(* IEC 61131-3 sources: com.logicals.lc3.webinar/usRTS_RPMControl_iSOC/src_FB_LIB_SAFE/Safe/PLCOpen (part 3) *)

(* ---- SF_PSE.iecst ---- *)
USING logicals.web.standard.safe;

NAMESPACE logicals.web.standard.safe
NAMESPACE plcopen

/*
 * This function block is a safety-related function block for monitoring Pressure-Sensitive-Equipment (PSE) like Safety Mats, Bumper etc.
 */
FUNCTION_BLOCK SF_PSE
	{ altName:="SF_PSE"; bgColor:="Gold"; width:=320; }
	VAR_INPUT
		/* See Section 5.1.1 General Input Parameters */
		Activate : BOOL := FALSE;
		/* Safety demand input.
		 * Variable.
		 * FALSE: PSE actuated, demand for safety-related response.
		 * TRUE: PSE not actuated, no demand for safety-related response.
		 * Safety control system must be able to detect a very short interruption of the PSE
		 * (which is specified in EN 1760: minimum 200 ms), when the PSE is used in applications as a safety device.
		 */
		S_PSE_In : SAFEBOOL := SAFEBOOL_Constant#SAFEFALSE;
		/* See Section 5.1.1 General Input Parameters */
		S_StartReset : SAFEBOOL := SAFEBOOL_Constant#SAFEFALSE;
		/* See Section 5.1.1 General Input Parameters */
		S_AutoReset : SAFEBOOL := SAFEBOOL_Constant#SAFEFALSE;
		/* See Section 5.1.1 General Input Parameters */
		Reset : BOOL := FALSE;
	END_VAR
	VAR_OUTPUT
		/* See Section 5.1.2 General Output Parameters */
		Ready : BOOL := FALSE;
		/* Output for the safety-related response.
		 * FALSE: Safety output disabled. Demand for safety-related response (e.g., reset requested or internal errors active).
		 * TRUE: Safety output enabled. No demand for safety-related response.
		 */
		S_PSE_Out : SAFEBOOL := SAFEBOOL_Constant#SAFEFALSE;
		/* Optional. See 5.1.2 General Output Parameters */
		SafetyDemand : BOOL := FALSE;
		/* Optional. See 5.1.2 General Output Parameters */
		ResetRequest : BOOL := FALSE;
		/* See Section 5.1.2 General Output Parameters */
		Error : BOOL := FALSE;
		/* See Section 5.1.2 General Output Parameters */
		DiagCode : WORD := 16#0000;
	END_VAR
	VAR
		GenericSafetyDemand : SFB_GenericSafetyDemand;
	END_VAR

	GenericSafetyDemand(
		Activate := Activate,
		S_SafetyDemandIn := S_PSE_In,
		S_StartReset := S_StartReset,
		S_AutoReset := S_AutoReset,
		Reset := Reset,
		Ready => Ready,
		S_SafetyDemandOut => S_PSE_Out,
		SafetyDemand => SafetyDemand,
		ResetRequest => ResetRequest,
		Error => Error,
		DiagCode => DiagCode,
		ENO => ENO
	);

END_FUNCTION_BLOCK

END_NAMESPACE
END_NAMESPACE

(* ---- SF_ResetButton.iecst ---- *)
USING logicals.web.standard.safe;

NAMESPACE logicals.web.standard.safe
NAMESPACE plcopen

TYPE
	SF_ResetButton_State : UINT(
	/* TrailingMinimum > TrailingMaximum OR TrailingMinimum < 100 msec. */
	Parameter_Error := 16#C000,
	/* ResetIn is TRUE while waiting for NOT ResetIn. */
	Reset_Error := 16#C001,
	/* TrailingMaximum elapsed before detecting F_TRIG at ResetIn. Waiting for R_TRIG at ResetIn. */
	Error_Trailing_Maximum := 16#C3E0,
	/* F_TRIG at ResetIn detected before TrailingMinimum elapsed. Waiting for R_TRIG at ResetIn. */
	Error_Trailing_Minimum := 16#C3F0,
	/* The function block is not active (initial state). */
	Idle := 16#0000,
	/* The function block is enabled. Wait for R_TRIG at ResetIn. */
	Wait_for_R_TRIG := 16#83E2,
	/* ResetIn is TRUE. Wait for F_TRIG at ResetIn */
	Wait_for_F_TRIG := 16#83F2,
	/* Valid reset behavior was detected. The state is valid for at least one cycle and will automatically transfer to 83E2. */
	Reset_Detected := 16#8000
	);
END_TYPE

/*
 * This function block adds the trailing edge functionality to all the function blocks with reset input with rising edge detection. This can be used to comply to EN ISO 13849-1:2015
 */
FUNCTION_BLOCK SF_ResetButton
	{ altName:="SF_ResetButton"; bgColor:="Gold"; width:=380; }
	VAR_INPUT
		/* Input which should be connected to the ResetRequest output of the paired FB.
			TRUE: ResetRequested
			FALSE: No reset requested / no monitoring of ResetIn. */
		ResetRequested : BOOL := TRUE;
		/* Variable.
			Input of reset button
			FALSE: reset button released;
			TRUE: reset button actuated by operator. */
		Button : BOOL := FALSE;
		/* Constant. Valid in trailing mode. Minimum time that the reset switch has to be actuated.
			If the reset button is pushed shorter than this time, the reset is ignored.
			Typical value 350msec.Absolut minimum value is 100msec.Minimum value 2 PLC cycles. */
		TrailingMinimum : TIME := T#350ms;
		/* Constant. Valid in trailing mode.
			Maximum time that the reset switch is actuated.
			Typical value can be around 2 sec. If the reset button is pushed longer than this time, the reset is ignored. */
		TrailingMaximum : TIME := T#2s;
	END_VAR
	VAR_OUTPUT
		/* See 5.1.2 General Output Parameters */
		Ready : BOOL := FALSE;
		/* Pulse for the initiation of the reset procedure.
			This pulse is generated after the falling edge.
			Pulse output with rising edge first. At least 1 cycle. */
		ResetOut : BOOL := FALSE;
		/* See 5.1.2 General Output Parameters */
		Error : BOOL := FALSE;
		/* See 5.1.2 General Output Parameters */
		DiagCode : WORD := 16#0000;
	END_VAR
	VAR
		TrailingMinimumTimer : TON;
		TrailingMaximumTimer : TON;
		R_Trig_Button : R_TRIG;
		F_Trig_Button : F_TRIG;
	END_VAR

	R_Trig_Button(Button);
	F_Trig_Button(Button);

	IF(NOT ResetRequested) THEN
		DiagCode := TO_WORD(SF_ResetButton_State#Idle);
	ELSE
		CASE TO_UINT(DiagCode) OF
			SF_ResetButton_State#Idle:
				/* IF(ResetRequested) THEN - ResetRequested is always true here */
					IF(Button) THEN
						DiagCode := TO_WORD(SF_ResetButton_State#Reset_Error);
					ELSE
					DiagCode := TO_WORD(SF_ResetButton_State#Wait_for_R_TRIG);
					END_IF;
			SF_ResetButton_State#Wait_for_R_TRIG:
				IF(TrailingMinimum > TrailingMaximum) OR (TrailingMinimum < T#100ms) THEN
					DiagCode := TO_WORD(SF_ResetButton_State#Parameter_Error);
				ELSIF(R_Trig_Button.Q) THEN
					DiagCode := TO_WORD(SF_ResetButton_State#Wait_for_F_TRIG);
				END_IF;
			SF_ResetButton_State#Reset_Error:
				IF(NOT Button) THEN
					DiagCode := TO_WORD(SF_ResetButton_State#Wait_for_R_TRIG);
				END_IF;
			SF_ResetButton_State#Wait_for_F_TRIG:
				TrailingMinimumTimer();
				TrailingMaximumTimer();
				IF(F_Trig_Button.Q) AND (NOT TrailingMinimumTimer.Q) THEN
					DiagCode := TO_WORD(SF_ResetButton_State#Error_Trailing_Minimum);
				ELSIF(TrailingMaximumTimer.Q) THEN
					DiagCode := TO_WORD(SF_ResetButton_State#Error_Trailing_Maximum);
				ELSIF(F_Trig_Button.Q) THEN
					DiagCode := TO_WORD(SF_ResetButton_State#Reset_Detected);
				END_IF;
			SF_ResetButton_State#Error_Trailing_Maximum:
				IF(R_Trig_Button.Q) THEN
					DiagCode := TO_WORD(SF_ResetButton_State#Wait_for_F_TRIG);
				END_IF;
			SF_ResetButton_State#Error_Trailing_Minimum:
				IF(R_Trig_Button.Q) THEN
					DiagCode := TO_WORD(SF_ResetButton_State#Wait_for_F_TRIG);
				END_IF;
			SF_ResetButton_State#Reset_Detected:
				DiagCode := TO_WORD(SF_ResetButton_State#Wait_for_R_TRIG);
			ELSE
				ENO := FALSE;
		END_CASE;
	END_IF;

		CASE TO_UINT(DiagCode) OF
			SF_ResetButton_State#Parameter_Error:
				TrailingMinimumTimer(IN := FALSE);
				TrailingMaximumTimer(IN := FALSE);
				Ready := TRUE;
				ResetOut := FALSE;
				Error := TRUE;
			SF_ResetButton_State#Reset_Error:
				TrailingMinimumTimer(IN := FALSE);
				TrailingMaximumTimer(IN := FALSE);
				Ready := TRUE;
				ResetOut := FALSE;
				Error := TRUE;
			SF_ResetButton_State#Error_Trailing_Maximum:
				TrailingMinimumTimer(IN := FALSE);
				TrailingMaximumTimer(IN := FALSE);
				Ready := TRUE;
				ResetOut := FALSE;
				Error := TRUE;
			SF_ResetButton_State#Error_Trailing_Minimum:
				TrailingMinimumTimer(IN := FALSE);
				TrailingMaximumTimer(IN := FALSE);
				Ready := TRUE;
				ResetOut := FALSE;
				Error := TRUE;
			SF_ResetButton_State#Idle:
				TrailingMinimumTimer(IN := FALSE);
				TrailingMaximumTimer(IN := FALSE);
				Ready := FALSE;
				ResetOut := FALSE;
				Error := FALSE;
			SF_ResetButton_State#Wait_for_R_TRIG:
				TrailingMinimumTimer(IN := FALSE);
				TrailingMaximumTimer(IN := FALSE);
				Ready := TRUE;
				ResetOut := FALSE;
				Error := FALSE;
			SF_ResetButton_State#Wait_for_F_TRIG:
				TrailingMinimumTimer(IN := TRUE, PT := TrailingMinimum);
				TrailingMaximumTimer(IN := TRUE, PT := TrailingMaximum);
				Ready := TRUE;
				ResetOut := FALSE;
				Error := FALSE;
			SF_ResetButton_State#Reset_Detected:
				TrailingMinimumTimer(IN := FALSE);
				TrailingMaximumTimer(IN := FALSE);
				Ready := TRUE;
				ResetOut := TRUE;
				Error := FALSE;
			ELSE
				ENO := FALSE;
		END_CASE;
END_FUNCTION_BLOCK

END_NAMESPACE
END_NAMESPACE

(* ---- SF_SafetyRequest.iecst ---- *)
USING logicals.web.standard.safe;

NAMESPACE logicals.web.standard.safe
NAMESPACE plcopen

TYPE
	SF_SafetyRequest_State : UINT(
	/* Acknowledgment lost while in the Safe state. */
	Acknowledge_Lost := 16#C010,
	/* S_OpMode request could not be completed within the monitoring time. */
	MonitoringTime_Elapsed := 16#C020,
	/* Static Reset detected in state 8401 (Init). */
	Reset_Error_1 := 16#C001,
	/* Static Reset detected in state C010 (Acknowledge Lost). */
	Reset_Error_2 := 16#C014,
	/* Static Reset detected in state C020 (MonitoringTime Elapsed). */
	Reset_Error_3 := 16#C011,
	/* The function block is not active (initial state). */
	Idle := 16#0000,
	/* Actuator is in a safe mode. */
	Safe_Mode:= 16#8000,
	/* State after Activate is set to TRUE or after a rising trigger at Reset. */
	Init := 16#8401,
	/* Operation mode without Acknowledge of safe mode */
	Operation_Mode:= 16#8802,
	/* Operation mode with Acknowledge of safe mode */
	Wait_For_Confirmation_OpMode := 16#8804,
	/* Waiting for confirmation from the drive (system interface). */
	Wait_For_Confirmation := 16#8002,
	/* Error was removed.
	* However S_OpMode must be set to TRUE or S_Acknowledge must become TRUE before the FB can be continued. */
	Wait_For_OpMode := 16#8004
	);
END_TYPE

/*
 * This function block provides the interface to a generic actuator, e.g. a safety drive or safety valve, to place the actuator in a safe state.
 */
FUNCTION_BLOCK SF_SafetyRequest
	{ altName:="SF_SafetyRequest"; bgColor:="Gold"; width:=400; }
	VAR_INPUT
		/* See Section 5.1.1 General Input Parameters */
		Activate : BOOL := FALSE;
		/* Variable.
		 * Requested mode of a generic safe actuator.
		 * FALSE: Safe mode is requested.
		 * TRUE: Operation mode is requested. */
		S_OpMode : SAFEBOOL := SAFEBOOL_Constant#SAFEFALSE;
		/* Variable.
		 * Confirmation of the generic actuator, if actuator is in the Safe state.
		 * FALSE: Operation mode (non-safe).
		 * TRUE: Safe mode. */
		S_Acknowledge : SAFEBOOL := SAFEBOOL_Constant#SAFEFALSE;
		/* Constant.
		 * Monitoring of the response time between the safety function request (S_OpMode set to FALSE)
		 * and the actuator acknowledgment (S_Acknowledge switches to TRUE). */
		MonitoringTime : TIME := T#0s;
		/* See Section 5.1.1 General Input Parameters */
		S_StartReset : SAFEBOOL := SAFEBOOL_Constant#SAFEFALSE;
		/* See Section 5.1.1 General Input Parameters with the functionality as an error removed acknowledge */
		Reset : BOOL := FALSE;
	END_VAR

	VAR_OUTPUT
		/* See Section 5.1.2 General Output Parameters */
		Ready : BOOL := FALSE;
		/* Confirmation of the Safe state.
		 * FALSE: Non-safe state.
		 * TRUE: Safe state. */
		S_SafetyActive : SAFEBOOL := SAFEBOOL_Constant#SAFEFALSE;
		/* Request to place the actuator in a safe state.
		 * FALSE: Safe state is requested.
		 * TRUE: Non-safe state. */
		S_SafetyRequest : SAFEBOOL := SAFEBOOL_Constant#SAFEFALSE;
		/* See Section 5.1.2 General Output Parameters */
		SafetyDemand : BOOL := FALSE;
		/* See Section 5.1.2 General Output Parameters */
		ResetRequest : BOOL := FALSE;
		/* See Section 5.1.2 General Output Parameters */
		Error : BOOL := FALSE;
		/* See Section 5.1.2 General Output Parameters */
		DiagCode : WORD := 16#0000;
	END_VAR

	VAR
		MonitoringTimer : TON;
		R_Trig_Reset : R_TRIG;
	END_VAR

	R_Trig_Reset(Reset);

	IF(NOT Activate) THEN
		DiagCode := TO_WORD(SF_SafetyRequest_State#Idle);
	ELSE
		CASE TO_UINT(DiagCode) OF
			SF_SafetyRequest_State#Idle:
				/* IF(Activate) THEN - ResetRequested is always true here */
					DiagCode := TO_WORD(SF_SafetyRequest_State#Init);
			SF_SafetyRequest_State#Init:
				IF(Reset AND NOT R_Trig_Reset.Q) THEN
					DiagCode := TO_WORD(SF_SafetyRequest_State#Reset_Error_1);
				ELSIF(R_Trig_Reset.Q AND IS_NOT(S_Acknowledge)) THEN
					DiagCode := TO_WORD(SF_SafetyRequest_State#Operation_Mode);
				ELSIF(R_Trig_Reset.Q AND IS(S_Acknowledge)) THEN
					DiagCode := TO_WORD(SF_SafetyRequest_State#Wait_For_Confirmation_OpMode);
				END_IF;
			SF_SafetyRequest_State#Operation_Mode:
				IF(IS_NOT(S_OpMode)) THEN
					DiagCode := TO_WORD(SF_SafetyRequest_State#Wait_For_Confirmation);
				ELSIF(IS(S_Acknowledge)) THEN
					DiagCode := TO_WORD(SF_SafetyRequest_State#Wait_For_Confirmation_OpMode);
				END_IF;
			SF_SafetyRequest_State#Wait_For_Confirmation_OpMode:
				IF(IS_NOT(S_Acknowledge)) THEN
					DiagCode := TO_WORD(SF_SafetyRequest_State#Operation_Mode);
				ELSIF(IS_NOT(S_OpMode)) THEN
					DiagCode := TO_WORD(SF_SafetyRequest_State#Wait_For_Confirmation);
				END_IF;
			SF_SafetyRequest_State#Wait_For_Confirmation:
				MonitoringTimer();
				IF(MonitoringTimer.Q) THEN
					DiagCode := TO_WORD(SF_SafetyRequest_State#MonitoringTime_Elapsed);
				ELSIF(IS(S_OpMode)) THEN
					DiagCode := TO_WORD(SF_SafetyRequest_State#Wait_For_Confirmation_OpMode);
				ELSIF(IS(S_Acknowledge)) THEN
					DiagCode := TO_WORD(SF_SafetyRequest_State#Safe_Mode);
				END_IF;
			SF_SafetyRequest_State#MonitoringTime_Elapsed:
				IF(Reset AND NOT R_Trig_Reset.Q) THEN
					DiagCode := TO_WORD(SF_SafetyRequest_State#Reset_Error_3);
				ELSIF(R_Trig_Reset.Q) THEN
					DiagCode := TO_WORD(SF_SafetyRequest_State#Wait_For_OpMode);
				END_IF;
			SF_SafetyRequest_State#Wait_For_OpMode:
				IF(IS(S_OpMode)) THEN
					DiagCode := TO_WORD(SF_SafetyRequest_State#Wait_For_Confirmation_OpMode);
				END_IF;
			SF_SafetyRequest_State#Safe_Mode:
				IF(IS_NOT(S_Acknowledge)) THEN
					DiagCode := TO_WORD(SF_SafetyRequest_State#Acknowledge_Lost);
				ELSIF(IS(S_OpMode)) THEN
					DiagCode := TO_WORD(SF_SafetyRequest_State#Wait_For_Confirmation_OpMode);
				END_IF;
			SF_SafetyRequest_State#Acknowledge_Lost:
				IF(Reset AND NOT R_Trig_Reset.Q) THEN
					DiagCode := TO_WORD(SF_SafetyRequest_State#Reset_Error_2);
				ELSIF(R_Trig_Reset.Q) THEN
					DiagCode := TO_WORD(SF_SafetyRequest_State#Wait_For_OpMode);
				END_IF;
			SF_SafetyRequest_State#Reset_Error_1:
				IF(NOT Reset) THEN
					DiagCode := TO_WORD(SF_SafetyRequest_State#Init);
				END_IF;
			SF_SafetyRequest_State#Reset_Error_2:
				IF(NOT Reset) THEN
					DiagCode := TO_WORD(SF_SafetyRequest_State#Acknowledge_Lost);
				END_IF;
			SF_SafetyRequest_State#Reset_Error_3:
				IF(NOT Reset) THEN
					DiagCode := TO_WORD(SF_SafetyRequest_State#MonitoringTime_Elapsed);
				END_IF;
		END_CASE;
	END_IF;

	CASE TO_UINT(DiagCode) OF
		SF_SafetyRequest_State#Idle:
			MonitoringTimer(IN := FALSE);
			Ready := FALSE;
			S_SafetyActive := SAFEBOOL_Constant#SAFEFALSE;
			S_SafetyRequest := SAFEBOOL_Constant#SAFEFALSE;
			SafetyDemand := FALSE;
			ResetRequest := FALSE;
			Error := FALSE;
		SF_SafetyRequest_State#Safe_Mode:
			MonitoringTimer(IN := FALSE);
			Ready := TRUE;
			S_SafetyActive := SAFEBOOL_Constant#SAFETRUE;
			S_SafetyRequest := SAFEBOOL_Constant#SAFEFALSE;
			SafetyDemand := FALSE;
			ResetRequest := FALSE;
			Error := FALSE;
		SF_SafetyRequest_State#Init:
			MonitoringTimer(IN := FALSE);
			Ready := TRUE;
			S_SafetyActive := SAFEBOOL_Constant#SAFEFALSE;
			S_SafetyRequest := SAFEBOOL_Constant#SAFEFALSE;
			SafetyDemand := FALSE;
			ResetRequest := TRUE;
			Error := FALSE;
		SF_SafetyRequest_State#Operation_Mode:
			MonitoringTimer(IN := FALSE);
			Ready := TRUE;
			S_SafetyActive := SAFEBOOL_Constant#SAFEFALSE;
			S_SafetyRequest := SAFEBOOL_Constant#SAFETRUE;
			SafetyDemand := TRUE;
			ResetRequest := FALSE;
			Error := FALSE;
		SF_SafetyRequest_State#Wait_For_Confirmation_OpMode:
			MonitoringTimer(IN := TRUE, PT := MonitoringTime);
			Ready := TRUE;
			S_SafetyActive := SAFEBOOL_Constant#SAFEFALSE;
			S_SafetyRequest := SAFEBOOL_Constant#SAFETRUE;
			SafetyDemand := TRUE;
			ResetRequest := FALSE;
			Error := FALSE;
		SF_SafetyRequest_State#Wait_For_Confirmation,
		SF_SafetyRequest_State#Wait_For_OpMode:
			MonitoringTimer(IN := TRUE, PT := MonitoringTime);
			Ready := TRUE;
			S_SafetyActive := SAFEBOOL_Constant#SAFEFALSE;
			S_SafetyRequest := SAFEBOOL_Constant#SAFEFALSE;
			SafetyDemand := FALSE;
			ResetRequest := FALSE;
			Error := FALSE;
		SF_SafetyRequest_State#Acknowledge_Lost,
		SF_SafetyRequest_State#MonitoringTime_Elapsed:
			MonitoringTimer(IN := FALSE);
			Ready := TRUE;
			S_SafetyActive := SAFEBOOL_Constant#SAFEFALSE;
			S_SafetyRequest := SAFEBOOL_Constant#SAFEFALSE;
			SafetyDemand := FALSE;
			ResetRequest := TRUE;
			Error := TRUE;
		SF_SafetyRequest_State#Reset_Error_1,
		SF_SafetyRequest_State#Reset_Error_2,
		SF_SafetyRequest_State#Reset_Error_3:
			MonitoringTimer(IN := FALSE);
			Ready := TRUE;
			S_SafetyActive := SAFEBOOL_Constant#SAFEFALSE;
			S_SafetyRequest := SAFEBOOL_Constant#SAFEFALSE;
			SafetyDemand := FALSE;
			ResetRequest := FALSE;
			Error := TRUE;
		ELSE
			ENO := FALSE;
	END_CASE;

	ENO := ENO AND CheckSAFEBOOL(S_OpMode) AND CheckSAFEBOOL(S_Acknowledge) AND CheckSAFEBOOL(S_StartReset);

END_FUNCTION_BLOCK

END_NAMESPACE
END_NAMESPACE

(* ---- SF_TestableSafetySensor.iecst ---- *)
USING logicals.web.standard.safe;

NAMESPACE logicals.web.standard.safe
NAMESPACE plcopen

TYPE
	SF_TestableSafetySensor_State : UINT(
	/* Invalid value at the TestTime parameter. Values between 0 ms and 150 ms are possible. */
	Parameter_Error := 16#C000,
	/* Static Reset condition detected after FB activation. */
	Reset_Error_1 := 16#C001,
	/* Static Reset condition detected in state 8403. */
	Reset_Error_2 := 16#C011,
	/* Static Reset condition detected in state Cx10. */
	Reset_Error_3 := 16#C021,
	/* Static Reset condition detected in state 8406. */
	Reset_Error_4 := 16#C031,
	/* Static Reset condition detected in state C000. */
	Reset_Error_5 := 16#C041,
	/* Static Reset condition detected in state 8413. */
	Reset_Error_6 := 16#C051,
	/* Test time elapsed in state 8020 or 8030. IF S_OSSD_IN = TRUE AND NoExternalTest = TRUE THEN x=4 ELSE x=0; */
	Test_Error_1 := 16#C410,
	Test_Error_2 := 16#C010,
	/* The function block is not active (initial state). */
	Idle := 16#0000,
	/* An activation has been detected by the FB. */
	Init := 16#8401,
	/* The FB has detected a safety demand. The switch has not been automatically tested yet. */
	ESPE_Interrupted_1 := 16#8802,
	/* Wait for rising trigger of Reset after state 8802. */
	Wait_for_Reset_1 := 16#8402,
	/* The automatic sensor test was faulty. An external manual sensor test is necessary.
	 * The support for the necessary external manual sensor test has been activated at the FB (NoExternalTest = FALSE).
	 * A negative signal edge at the sensor is required.
	 */
	External_Function_Test := 16#8002,
	/* The automatic sensor test was faulty. An external manual sensor test is necessary.
	 * The support for the necessary external manual sensor test has been activated at the FB (NoExternalTest = FALSE).
	 * A TRUE signal at the sensor is required.
	 */
	ESPE_Interrupted_External_Test := 16#8804,
	/* The automatic sensor test was faulty. An external manual sensor test is necessary.
	 * The support for the necessary external manual sensor test has been activated at the FB (NoExternalTest = FALSE).
	 * The external manual test is complete. The FB detected a complete sensor switching cycle (external controlled).
	 */
	End_External_Test := 16#8404,
	/* The FB has not detected a safety demand. The sensor has not been tested automatically. */
	ESPE_Free_No_Test := 16#8010,
	/* The FB has detected a safety demand. The switch was automatically tested. */
	ESPE_Interrupted_2 := 16#8806,
	/* Wait for rising trigger of Reset after state 8812. */
	Wait_for_Reset_2 := 16#8406,
	/* The automatic sensor test is active. Test Timer is started first time. The transmitter signal of the sensor is switched off by the FB.
	 * The signal of the receiver must follow the signal of the transmitter.
	 */
	Test_Request := 16#8020,
	/* The automatic sensor test is active. Test Timer is started second time.
	 * The transmitter signal of the sensor is switched on by the FB. The signal of the receiver must follow the signal of the transmitter.
	 */
	Test_Active := 16#8030,
	/* The FB has not detected a safety demand. The sensor was automatically tested. */
	ESPE_Free_Test_ok := 16#8000
	);
END_TYPE

FUNCTION_BLOCK SF_TestableSafetySensor
	{ altName:="SF_TestableSafetySensor"; bgColor:="Gold"; width:=440;}
	VAR_INPUT
		/* See Section 5.1.1 General Input Parameters */
		Activate : BOOL := FALSE;
		/* Variable.
		 * Status of sensor output, e.g., light curtain.
		 * FALSE: Safety sensor in test state or demand for safety-related response.
		 * TRUE: Sensor in the state for normal operating conditions.
		 */
		S_OSSD_In : SAFEBOOL := SAFEBOOL_Constant#SAFEFALSE;
		/* Variable.
		 * Input to start sensor test. Sets "S_TestOut" and starts the internal time monitoring function in the FB.
		 * FALSE: No test requested.
		 * TRUE: Test requested.
		 */
		StartTest : BOOL := FALSE;
		/* Constant. Range: 0 ... 150ms. Test time of safety sensor. */
		TestTime : TIME := T#10ms;
		/* Constant.
		 * Indicates if external manual sensor test is supported.
		 * FALSE: The external manual sensor test is supported. Only after a complete manual sensor switching sequence, a automatic test is possible again after a faulty automatic sensor test.
		 * TRUE: The external manual sensor test is not supported.
		 * An automatic test is possible again without a manual sensor switching sequence after faulty automatic sensor test.
		 */
		NoExternalTest : BOOL := FALSE;
		/* See Section 5.1.1 General Input Parameters */
		S_StartReset : SAFEBOOL := SAFEBOOL_Constant#SAFEFALSE;
		/* See Section 5.1.1 General Input Parameters */
		S_AutoReset : SAFEBOOL := SAFEBOOL_Constant#SAFEFALSE;
		/* See Section 5.1.1 General Input Parameters */
		Reset : BOOL := FALSE;
	END_VAR
	VAR_OUTPUT
		/* See Section 5.1.2 General Output Parameters */
		Ready : BOOL := FALSE;
		/* Safety related output indicating the status of the ESPE.
		 * FALSE: The sensor has a safety-related action request or test error.
		 * TRUE: The sensor has no safety-related action request AND no test error.
		 */
		S_OSSD_Out : SAFEBOOL := SAFEBOOL_Constant#SAFEFALSE;
		/* Coupled with the test input of the sensor. Although specified as SAFEBOOL, in practice this signal will often be connected to a BOOL output.
		 * FALSE: Test request issued.
		 * TRUE: No test request.
		 */
		S_TestOut : SAFEBOOL := SAFEBOOL_Constant#SAFETRUE;
		/* Feedback signal to the process.
		 * FALSE: An automatic sensor test is not possible.
		 * TRUE: An automatic sensor test is possible.
		 */
		TestPossible : BOOL := FALSE;
		/* A positive signal edge indicates the successful execution of the automatic sensor test.
		 * FALSE:
		 * - An automatic sensor test was not executed yet.
		 * - An automatic sensor test is active.
		 * - An automatic sensor test was faulty.
		 * TRUE: A sensor test was executed successfully.
		 */
		TestExecuted : BOOL := FALSE;
		/* Optional. See 5.1.2 General Output Parameters */
		SafetyDemand : BOOL := FALSE;
		/* Optional. See 5.1.2 General Output Parameters */
		ResetRequest : BOOL := FALSE;
		/* See Section 5.1.2 General Output Parameters */
		Error : BOOL := FALSE;
		/* See Section 5.1.2 General Output Parameters */
		DiagCode : WORD := 16#0000;
	END_VAR
	VAR
		R_Trig_Reset : R_TRIG;
		R_Trig_S_OSSD_In : R_TRIG;
		R_Trig_StartTest : R_TRIG;
		F_Trig_S_OSSD_In : F_TRIG;
		Timer1 : TON;
		Timer2 : TON;
	END_VAR

	R_Trig_Reset(Reset);
	R_Trig_S_OSSD_In(IS(S_OSSD_In));
	R_Trig_StartTest(StartTest);
	F_Trig_S_OSSD_In(IS(S_OSSD_In));

	IF(NOT Activate) THEN
		DiagCode := TO_WORD(SF_TestableSafetySensor_State#Idle);
	ELSE
		CASE TO_UINT(DiagCode) OF
			SF_TestableSafetySensor_State#Idle:
				/* IF(Activate) THEN - Active is always true here */
					DiagCode := TO_WORD(SF_TestableSafetySensor_State#Init);
			SF_TestableSafetySensor_State#Init:
				IF(TestTime > T#150ms) THEN
					DiagCode := TO_WORD(SF_TestableSafetySensor_State#Parameter_Error);
				ELSIF(Reset AND NOT R_Trig_Reset.Q) THEN
					DiagCode := TO_WORD(SF_TestableSafetySensor_State#Reset_Error_1);
				ELSIF(IS_NOT(S_OSSD_In)) THEN
					DiagCode := TO_WORD(SF_TestableSafetySensor_State#ESPE_Interrupted_1);
				ELSIF(IS(S_OSSD_In) AND NOT R_Trig_S_OSSD_In.Q AND (R_Trig_Reset.Q OR IS(S_StartReset))) THEN
					DiagCode := TO_WORD(SF_TestableSafetySensor_State#ESPE_Free_No_Test);
				END_IF;
			SF_TestableSafetySensor_State#Parameter_Error:
				IF(Reset AND NOT R_Trig_Reset.Q) THEN
					DiagCode := TO_WORD(SF_TestableSafetySensor_State#Reset_Error_5);
				ELSIF(R_Trig_Reset.Q AND TestTime <= T#150ms) THEN
					DiagCode := TO_WORD(SF_TestableSafetySensor_State#Init);
				END_IF;
			SF_TestableSafetySensor_State#Reset_Error_5:
				IF(NOT Reset) THEN
					DiagCode := TO_WORD(SF_TestableSafetySensor_State#Parameter_Error);
				END_IF;
			SF_TestableSafetySensor_State#Reset_Error_1:
				IF(NOT Reset) THEN
					DiagCode := TO_WORD(SF_TestableSafetySensor_State#Init);
				END_IF;
			SF_TestableSafetySensor_State#ESPE_Interrupted_1:
				IF(IS(S_OSSD_In)) THEN
					DiagCode := TO_WORD(SF_TestableSafetySensor_State#Wait_for_Reset_1);
				END_IF;
			SF_TestableSafetySensor_State#End_External_Test:
				IF(Reset AND NOT R_Trig_Reset.Q) THEN
					DiagCode := TO_WORD(SF_TestableSafetySensor_State#Reset_Error_4);
				ELSIF(R_Trig_Reset.Q AND IS_NOT(S_OSSD_In)) THEN
					DiagCode := TO_WORD(SF_TestableSafetySensor_State#ESPE_Interrupted_1);
				ELSIF(R_Trig_Reset.Q AND IS(S_OSSD_In) AND NOT R_Trig_S_OSSD_In.Q) THEN
					DiagCode := TO_WORD(SF_TestableSafetySensor_State#ESPE_Free_No_Test);
				END_IF;
			SF_TestableSafetySensor_State#Reset_Error_4:
				IF(NOT Reset) THEN
					DiagCode := TO_WORD(SF_TestableSafetySensor_State#End_External_Test);
				END_IF;
			SF_TestableSafetySensor_State#ESPE_Interrupted_External_Test:
				IF(IS(S_OSSD_In)) THEN
					DiagCode := TO_WORD(SF_TestableSafetySensor_State#End_External_Test);
				END_IF;
			SF_TestableSafetySensor_State#External_Function_Test:
				IF(F_Trig_S_OSSD_In.Q) THEN
					DiagCode := TO_WORD(SF_TestableSafetySensor_State#ESPE_Interrupted_External_Test);
				END_IF;
			SF_TestableSafetySensor_State#Test_Request:
				IF(Timer1.Q AND IS(S_OSSD_In) AND NoExternalTest) THEN
					DiagCode := TO_WORD(SF_TestableSafetySensor_State#Test_Error_1);
				ELSIF(Timer1.Q) THEN
					DiagCode := TO_WORD(SF_TestableSafetySensor_State#Test_Error_2);
				ELSIF(IS_NOT(S_OSSD_In)) THEN
					DiagCode := TO_WORD(SF_TestableSafetySensor_State#Test_Active);
				END_IF;
			SF_TestableSafetySensor_State#Test_Active:
				IF(Timer2.Q AND IS(S_OSSD_In) AND NoExternalTest) THEN
						DiagCode := TO_WORD(SF_TestableSafetySensor_State#Test_Error_1);
				ELSIF(Timer2.Q) THEN
						DiagCode := TO_WORD(SF_TestableSafetySensor_State#Test_Error_2);
				ELSIF(IS(S_OSSD_In)) THEN
					DiagCode := TO_WORD(SF_TestableSafetySensor_State#ESPE_Free_Test_ok);
				END_IF;
			SF_TestableSafetySensor_State#Test_Error_1,
			SF_TestableSafetySensor_State#Test_Error_2:
				IF(Reset AND NOT R_Trig_Reset.Q) THEN
					DiagCode := TO_WORD(SF_TestableSafetySensor_State#Reset_Error_3);
				ELSIF(R_Trig_Reset.Q AND NOT NoExternalTest) THEN
					DiagCode := TO_WORD(SF_TestableSafetySensor_State#External_Function_Test);
				ELSIF(IS(S_OSSD_In) AND NOT R_Trig_S_OSSD_In.Q AND R_Trig_Reset.Q AND NoExternalTest) THEN
					DiagCode := TO_WORD(SF_TestableSafetySensor_State#ESPE_Free_No_Test);
				END_IF;
			SF_TestableSafetySensor_State#Reset_Error_3:
				IF(NOT Reset AND IS(S_OSSD_In) AND NoExternalTest) THEN
					DiagCode := TO_WORD(SF_TestableSafetySensor_State#Test_Error_1);
				ELSIF(NOT Reset) THEN
					DiagCode := TO_WORD(SF_TestableSafetySensor_State#Test_Error_2);
				END_IF;
			SF_TestableSafetySensor_State#Wait_for_Reset_1:
				IF(Reset AND NOT R_Trig_Reset.Q) THEN
					DiagCode := TO_WORD(SF_TestableSafetySensor_State#Reset_Error_2);
				ELSIF(IS_NOT(S_OSSD_In)) THEN
					DiagCode := TO_WORD(SF_TestableSafetySensor_State#ESPE_Interrupted_1);
				ELSIF(IS(S_OSSD_In) AND NOT R_Trig_S_OSSD_In.Q AND (R_Trig_Reset.Q OR IS(S_AutoReset))) THEN
					DiagCode := TO_WORD(SF_TestableSafetySensor_State#ESPE_Free_No_Test);
				END_IF;
			SF_TestableSafetySensor_State#Reset_Error_2:
				IF(NOT Reset) THEN
					DiagCode := TO_WORD(SF_TestableSafetySensor_State#Wait_for_Reset_1);
				END_IF;
			SF_TestableSafetySensor_State#ESPE_Free_No_Test:
				IF(IS_NOT(S_OSSD_In)) THEN
					DiagCode := TO_WORD(SF_TestableSafetySensor_State#ESPE_Interrupted_1);
				ELSIF(R_Trig_StartTest.Q) THEN
					DiagCode := TO_WORD(SF_TestableSafetySensor_State#Test_Request);
				END_IF;
			SF_TestableSafetySensor_State#ESPE_Free_Test_ok:
				IF(IS_NOT(S_OSSD_In)) THEN
					DiagCode := TO_WORD(SF_TestableSafetySensor_State#ESPE_Interrupted_2);
				ELSIF(R_Trig_StartTest.Q) THEN
					DiagCode := TO_WORD(SF_TestableSafetySensor_State#Test_Request);
				END_IF;
			SF_TestableSafetySensor_State#Wait_for_Reset_2:
				IF(Reset AND NOT R_Trig_Reset.Q) THEN
					DiagCode := TO_WORD(SF_TestableSafetySensor_State#Reset_Error_6);
				ELSIF(IS_NOT(S_OSSD_In)) THEN
					DiagCode := TO_WORD(SF_TestableSafetySensor_State#ESPE_Interrupted_2);
				ELSIF(IS(S_OSSD_In) AND (R_Trig_Reset.Q OR IS(S_AutoReset))) THEN
					DiagCode := TO_WORD(SF_TestableSafetySensor_State#ESPE_Free_Test_ok);
				END_IF;
			SF_TestableSafetySensor_State#Reset_Error_6:
				IF(NOT Reset) THEN
					DiagCode := TO_WORD(SF_TestableSafetySensor_State#Wait_for_Reset_2);
				END_IF;
			SF_TestableSafetySensor_State#ESPE_Interrupted_2:
				IF(IS(S_OSSD_In)) THEN
					DiagCode := TO_WORD(SF_TestableSafetySensor_State#Wait_for_Reset_2);
				END_IF;
			ELSE
				ENO := FALSE;
		END_CASE;
	END_IF;

	CASE TO_UINT(DiagCode) OF
		SF_TestableSafetySensor_State#Idle:
			Timer1(IN := FALSE);
			Timer2(IN := FALSE);
			Ready := FALSE;
			S_OSSD_Out := SAFEBOOL_Constant#SAFEFALSE;
			S_TestOut := SAFEBOOL_Constant#SAFETRUE;
			TestPossible := FALSE;
			TestExecuted := FALSE;
			SafetyDemand := FALSE;
			ResetRequest := FALSE;
			Error := FALSE;
		SF_TestableSafetySensor_State#Init,
		SF_TestableSafetySensor_State#Wait_for_Reset_1,
		SF_TestableSafetySensor_State#End_External_Test:
			Timer1(IN := FALSE);
			Timer2(IN := FALSE);
			Ready := TRUE;
			S_OSSD_Out := SAFEBOOL_Constant#SAFEFALSE;
			S_TestOut := SAFEBOOL_Constant#SAFETRUE;
			TestPossible := FALSE;
			TestExecuted := FALSE;
			SafetyDemand := FALSE;
			ResetRequest := TRUE;
			Error := FALSE;
		SF_TestableSafetySensor_State#ESPE_Interrupted_1,
		SF_TestableSafetySensor_State#ESPE_Interrupted_External_Test:
			Timer1(IN := FALSE);
			Timer2(IN := FALSE);
			Ready := TRUE;
			S_OSSD_Out := SAFEBOOL_Constant#SAFEFALSE;
			S_TestOut := SAFEBOOL_Constant#SAFETRUE;
			TestPossible := FALSE;
			TestExecuted := FALSE;
			SafetyDemand := TRUE;
			ResetRequest := FALSE;
			Error := FALSE;
		SF_TestableSafetySensor_State#ESPE_Interrupted_2:
			Timer1(IN := FALSE);
			Timer2(IN := FALSE);
			Ready := TRUE;
			S_OSSD_Out := SAFEBOOL_Constant#SAFEFALSE;
			S_TestOut := SAFEBOOL_Constant#SAFETRUE;
			TestPossible := FALSE;
			TestExecuted := TRUE;
			SafetyDemand := TRUE;
			ResetRequest := FALSE;
			Error := FALSE;
		SF_TestableSafetySensor_State#External_Function_Test:
			Timer1(IN := FALSE);
			Timer2(IN := FALSE);
			Ready := TRUE;
			S_OSSD_Out := SAFEBOOL_Constant#SAFEFALSE;
			S_TestOut := SAFEBOOL_Constant#SAFETRUE;
			TestPossible := FALSE;
			TestExecuted := FALSE;
			SafetyDemand := FALSE;
			ResetRequest := FALSE;
			Error := FALSE;
		SF_TestableSafetySensor_State#ESPE_Free_No_Test:
			Timer1(IN := FALSE);
			Timer2(IN := FALSE);
			Ready := TRUE;
			S_OSSD_Out := SAFEBOOL_Constant#SAFETRUE;
			S_TestOut := SAFEBOOL_Constant#SAFETRUE;
			TestPossible := TRUE;
			TestExecuted := FALSE;
			SafetyDemand := FALSE;
			ResetRequest := FALSE;
			Error := FALSE;
		SF_TestableSafetySensor_State#Wait_for_Reset_2:
			Timer1(IN := FALSE);
			Timer2(IN := FALSE);
			Ready := TRUE;
			S_OSSD_Out := SAFEBOOL_Constant#SAFEFALSE;
			S_TestOut := SAFEBOOL_Constant#SAFETRUE;
			TestPossible := FALSE;
			TestExecuted := TRUE;
			SafetyDemand := FALSE;
			ResetRequest := TRUE;
			Error := FALSE;
		SF_TestableSafetySensor_State#Test_Request:
			Timer1(IN := TRUE, PT := TestTime);
			Timer2(IN := FALSE);
			Ready := TRUE;
			S_OSSD_Out := SAFEBOOL_Constant#SAFETRUE;
			S_TestOut := SAFEBOOL_Constant#SAFEFALSE;
			TestPossible := FALSE;
			TestExecuted := FALSE;
			SafetyDemand := FALSE;
			ResetRequest := FALSE;
			Error := FALSE;
		SF_TestableSafetySensor_State#Test_Active:
			Timer1(IN := FALSE);
			Timer2(IN := TRUE, PT := TestTime);
			Ready := TRUE;
			S_OSSD_Out := SAFEBOOL_Constant#SAFETRUE;
			S_TestOut := SAFEBOOL_Constant#SAFETRUE;
			TestPossible := FALSE;
			TestExecuted := FALSE;
			SafetyDemand := FALSE;
			ResetRequest := FALSE;
			Error := FALSE;
		SF_TestableSafetySensor_State#ESPE_Free_Test_ok:
			Timer1(IN := FALSE);
			Timer2(IN := FALSE);
			Ready := TRUE;
			S_OSSD_Out := SAFEBOOL_Constant#SAFETRUE;
			S_TestOut := SAFEBOOL_Constant#SAFETRUE;
			TestPossible := TRUE;
			TestExecuted := TRUE;
			SafetyDemand := FALSE;
			ResetRequest := FALSE;
			Error := FALSE;
		SF_TestableSafetySensor_State#Parameter_Error,
		SF_TestableSafetySensor_State#Reset_Error_1,
		SF_TestableSafetySensor_State#Reset_Error_2,
		SF_TestableSafetySensor_State#Reset_Error_3,
		SF_TestableSafetySensor_State#Reset_Error_4,
		SF_TestableSafetySensor_State#Reset_Error_5:
			Timer1(IN := FALSE);
			Timer2(IN := FALSE);
			Ready := TRUE;
			S_OSSD_Out := SAFEBOOL_Constant#SAFEFALSE;
			S_TestOut := SAFEBOOL_Constant#SAFETRUE;
			TestPossible := FALSE;
			TestExecuted := FALSE;
			SafetyDemand := FALSE;
			ResetRequest := FALSE;
			Error := TRUE;
		SF_TestableSafetySensor_State#Reset_Error_6:
			Timer1(IN := FALSE);
			Timer2(IN := FALSE);
			Ready := TRUE;
			S_OSSD_Out := SAFEBOOL_Constant#SAFEFALSE;
			S_TestOut := SAFEBOOL_Constant#SAFETRUE;
			TestPossible := FALSE;
			TestExecuted := TRUE;
			SafetyDemand := FALSE;
			ResetRequest := FALSE;
			Error := TRUE;
		SF_TestableSafetySensor_State#Test_Error_1:
			Timer1(IN := FALSE);
			Timer2(IN := FALSE);
			Ready := TRUE;
			S_OSSD_Out := SAFEBOOL_Constant#SAFEFALSE;
			S_TestOut := SAFEBOOL_Constant#SAFETRUE;
			TestPossible := FALSE;
			TestExecuted := FALSE;
			SafetyDemand := FALSE;
			ResetRequest := TRUE;
			Error := TRUE;
		SF_TestableSafetySensor_State#Test_Error_2:
			Timer1(IN := FALSE);
			Timer2(IN := FALSE);
			Ready := TRUE;
			S_OSSD_Out := SAFEBOOL_Constant#SAFEFALSE;
			S_TestOut := SAFEBOOL_Constant#SAFETRUE;
			TestPossible := FALSE;
			TestExecuted := FALSE;
			SafetyDemand := FALSE;
			ResetRequest := FALSE;
			Error := TRUE;
		ELSE
			ENO := FALSE;
	END_CASE;

	ENO := ENO AND CheckSAFEBOOL(S_OSSD_In) AND CheckSAFEBOOL(S_StartReset) AND CheckSAFEBOOL(S_AutoReset);

END_FUNCTION_BLOCK

END_NAMESPACE
END_NAMESPACE

(* ---- SF_TwoHandControlTypeII.iecst ---- *)
USING logicals.web.standard.safe;

NAMESPACE logicals.web.standard.safe
NAMESPACE plcopen

TYPE
	SF_TwoHandControlTypeII_State : UINT(
	/* S_Button1 was TRUE on FB activation */
	Error_B1 := 16#C010,
	/* S_Button2 was TRUE on FB activation */
	Error_B2 := 16#C020,
	/* The signals at S_Button1 and S_Button2 were TRUE on FB activation */
	Error_B1_and_B2 := 16#C030,
	/* The function block is not active (initial state). */
	Idle := 16#0000,
	/* Both buttons actuated correctly. The safety related output is enabled. */
	Buttons_Actuated := 16#8000,
	/* Function block is active, but in init state. */
	Init := 16#8001,
	/* No button is actuated. */
	Buttons_Released := 16#8802,
	/* Only Button 1 is actuated */
	Button_1_Actuated := 16#8004,
	/* Only Button 2 is activated */
	Button_2_Actuated := 16#8806,
	/* The safety related output was enabled and is disabled again.
	 * FALSE at both S_Button1 and S_Button2 was not achieved after disa-bling the safety related output.
	 * In this state, S_Button1 is TRUE and S_Button2 is FALSE after disabling the safety related output.
	 */
	Button_2_Released := 16#8808,
	/* The safety related output was enabled and is disabled again.
	 * FALSE at both S_Button1 and S_Button2 was not achieved after disa-bling the safety related output.
	 * In this state, S_Button1 is FALSE and S_Button2 is TRUE after disabling the safety related output.
	 */
	Button_1_Released := 16#880A,
	/* The safety related output was enabled and is disabled again.
	 * FALSE at both S_Button1 and S_Button2 was not achieved after disa-bling the safety related output.
	 * In this state, S_Button1 is TRUE and S_Button2 is TRUE after disabling the safety related output.
	 */
	Locked_Off := 16#880C,
	/* Incorrect actuation of the buttons. Waiting for release of both buttons */
	Locked_On := 16#880E
	);
END_TYPE

/*
 * This function block provides the two-hand control functionality (see EN 574, Section 4 Type II).
 */
FUNCTION_BLOCK SF_TwoHandControlTypeII
	{ altName:="SF_TwoHandControlTypeII"; bgColor:="Gold"; width:=420; }
	VAR_INPUT
		/* See Section 5.1.1 General Input Parameters */
		Activate : BOOL := FALSE;
		/* Variable.
		 * Input of button 1 )
		 * FALSE: Button 1 released.
		 * TRUE: Button 1 actuated. */
		S_Button1 : SAFEBOOL := SAFEBOOL_Constant#SAFEFALSE;
		/* Variable.
		 * Input of button 2 )
		 * FALSE: Button 2 released.
		 * TRUE: Button 2 actuated. */
		S_Button2 : SAFEBOOL := SAFEBOOL_Constant#SAFEFALSE;
	END_VAR
	VAR_OUTPUT
		/* See Section 5.1.2 General Output Parameters */
		Ready : BOOL := FALSE;
		/* Safety related output signal.
		 * FALSE: No correct two hand operation.
		 * TRUE: S_Button1 and S_Button2 inputs are TRUE and no error occurred. Correct two hand operation. */
		S_TwoHandOut : SAFEBOOL := FALSE;
		/* Optional. See 5.1.2 General Output Parameters */
		SafetyDemand : BOOL := FALSE;
		/* See Section 5.1.2 General Output Parameters */
		Error : BOOL := FALSE;
		/* See Section 5.1.2 General Output Parameters */
		DiagCode : WORD := 16#0000;
	END_VAR

	IF(NOT Activate) THEN
		DiagCode := TO_WORD(SF_TwoHandControlTypeII_State#Idle);
	ELSE
		CASE TO_UINT(DiagCode) OF
			SF_TwoHandControlTypeII_State#Idle:
				/* IF(Activate) THEN - Active is always true here */
					DiagCode := TO_WORD(SF_TwoHandControlTypeII_State#Init);
			SF_TwoHandControlTypeII_State#Init:
				IF(IS(S_Button1)) AND (IS_NOT(S_Button2)) THEN
					DiagCode := TO_WORD(SF_TwoHandControlTypeII_State#Error_B1);
				ELSIF(IS(S_Button2)) AND (IS_NOT(S_Button1)) THEN
					DiagCode := TO_WORD(SF_TwoHandControlTypeII_State#Error_B2);
				ELSIF(IS(S_Button1)) AND (IS(S_Button2)) THEN
					DiagCode := TO_WORD(SF_TwoHandControlTypeII_State#Error_B1_and_B2);
				ELSE /* (IS_NOT(S_Button1)) AND (IS_NOT(S_Button2)) THEN */
					DiagCode := TO_WORD(SF_TwoHandControlTypeII_State#Buttons_Released);
				END_IF;
			SF_TwoHandControlTypeII_State#Error_B1:
				IF(IS_NOT(S_Button1)) AND (IS_NOT(S_Button2)) THEN
					DiagCode := TO_WORD(SF_TwoHandControlTypeII_State#Buttons_Released);
				END_IF;
			SF_TwoHandControlTypeII_State#Error_B2:
				IF(IS_NOT(S_Button1)) AND (IS_NOT(S_Button2)) THEN
					DiagCode := TO_WORD(SF_TwoHandControlTypeII_State#Buttons_Released);
				END_IF;
			SF_TwoHandControlTypeII_State#Error_B1_and_B2:
				IF(IS_NOT(S_Button1)) AND (IS_NOT(S_Button2)) THEN
					DiagCode := TO_WORD(SF_TwoHandControlTypeII_State#Buttons_Released);
				END_IF;
			SF_TwoHandControlTypeII_State#Buttons_Released:
				IF(IS(S_Button1)) AND (IS(S_Button2)) THEN
					DiagCode := TO_WORD(SF_TwoHandControlTypeII_State#Buttons_Actuated);
				ELSIF(IS(S_Button1)) THEN
					DiagCode := TO_WORD(SF_TwoHandControlTypeII_State#Button_1_Actuated);
				ELSIF(IS(S_Button2)) THEN
					DiagCode := TO_WORD(SF_TwoHandControlTypeII_State#Button_2_Actuated);
				END_IF;
			SF_TwoHandControlTypeII_State#Button_1_Actuated:
				IF(IS_NOT(S_Button1)) AND (IS_NOT(S_Button2)) THEN
					DiagCode := TO_WORD(SF_TwoHandControlTypeII_State#Buttons_Released);
				ELSIF(IS_NOT(S_Button1)) AND (IS(S_Button2)) THEN
					DiagCode := TO_WORD(SF_TwoHandControlTypeII_State#Locked_On);
				ELSIF(IS(S_Button1)) AND (IS(S_Button2)) THEN
					DiagCode := TO_WORD(SF_TwoHandControlTypeII_State#Buttons_Actuated);
				END_IF;
			SF_TwoHandControlTypeII_State#Locked_On:
				IF(IS_NOT(S_Button1)) AND (IS_NOT(S_Button2)) THEN
					DiagCode := TO_WORD(SF_TwoHandControlTypeII_State#Buttons_Released);
				END_IF;
			SF_TwoHandControlTypeII_State#Button_2_Actuated:
				IF(IS_NOT(S_Button1)) AND (IS_NOT(S_Button2)) THEN
					DiagCode := TO_WORD(SF_TwoHandControlTypeII_State#Buttons_Released);
				ELSIF(IS(S_Button1)) AND (IS_NOT(S_Button2)) THEN
					DiagCode := TO_WORD(SF_TwoHandControlTypeII_State#Locked_On);
				ELSIF(IS(S_Button1)) AND (IS(S_Button2)) THEN
					DiagCode := TO_WORD(SF_TwoHandControlTypeII_State#Buttons_Actuated);
				END_IF;
			SF_TwoHandControlTypeII_State#Locked_Off:
				IF(IS_NOT(S_Button1)) AND (IS(S_Button2)) THEN
					DiagCode := TO_WORD(SF_TwoHandControlTypeII_State#Button_1_Released);
				ELSIF(IS(S_Button1)) AND (IS_NOT(S_Button2)) THEN
					DiagCode := TO_WORD(SF_TwoHandControlTypeII_State#Button_2_Released);
				ELSIF(IS_NOT(S_Button1)) AND (IS_NOT(S_Button2)) THEN
					DiagCode := TO_WORD(SF_TwoHandControlTypeII_State#Buttons_Released);
				END_IF;
			SF_TwoHandControlTypeII_State#Button_1_Released:
				IF(IS(S_Button1)) AND (IS(S_Button2)) THEN
					DiagCode := TO_WORD(SF_TwoHandControlTypeII_State#Locked_Off);
				ELSIF(IS(S_Button1)) AND (IS_NOT(S_Button2)) THEN
					DiagCode := TO_WORD(SF_TwoHandControlTypeII_State#Button_2_Released);
				ELSIF(IS_NOT(S_Button1)) AND (IS_NOT(S_Button2)) THEN
					DiagCode := TO_WORD(SF_TwoHandControlTypeII_State#Buttons_Released);
				END_IF;
			SF_TwoHandControlTypeII_State#Button_2_Released:
				IF(IS(S_Button1)) AND (IS(S_Button2)) THEN
					DiagCode := TO_WORD(SF_TwoHandControlTypeII_State#Locked_Off);
				ELSIF(IS_NOT(S_Button1)) AND (IS(S_Button2)) THEN
					DiagCode := TO_WORD(SF_TwoHandControlTypeII_State#Button_1_Released);
				ELSIF(IS_NOT(S_Button1)) AND (IS_NOT(S_Button2)) THEN
					DiagCode := TO_WORD(SF_TwoHandControlTypeII_State#Buttons_Released);
				END_IF;
			SF_TwoHandControlTypeII_State#Buttons_Actuated:
				IF(IS(S_Button1)) AND (IS_NOT(S_Button2)) THEN
					DiagCode := TO_WORD(SF_TwoHandControlTypeII_State#Button_2_Released);
				ELSIF(IS_NOT(S_Button1)) AND (IS(S_Button2)) THEN
					DiagCode := TO_WORD(SF_TwoHandControlTypeII_State#Button_1_Released);
				ELSIF(IS_NOT(S_Button1)) AND (IS_NOT(S_Button2)) THEN
					DiagCode := TO_WORD(SF_TwoHandControlTypeII_State#Buttons_Released);
				END_IF;
			ELSE
				ENO := FALSE;
		END_CASE;
	END_IF;

	CASE TO_UINT(DiagCode) OF
		SF_TwoHandControlTypeII_State#Idle:
			Ready := FALSE;
			S_TwoHandOut := SAFEBOOL_Constant#SAFEFALSE;
			SafetyDemand := FALSE;
			Error := FALSE;
		SF_TwoHandControlTypeII_State#Buttons_Actuated:
			Ready := TRUE;
			S_TwoHandOut := SAFEBOOL_Constant#SAFETRUE;
			SafetyDemand := FALSE;
			Error := FALSE;
		SF_TwoHandControlTypeII_State#Init:
			Ready := TRUE;
			S_TwoHandOut := SAFEBOOL_Constant#SAFEFALSE;
			SafetyDemand := FALSE;
			Error := FALSE;
		SF_TwoHandControlTypeII_State#Buttons_Released,
		SF_TwoHandControlTypeII_State#Button_1_Actuated,
		SF_TwoHandControlTypeII_State#Button_2_Actuated,
		SF_TwoHandControlTypeII_State#Button_2_Released,
		SF_TwoHandControlTypeII_State#Button_1_Released,
		SF_TwoHandControlTypeII_State#Locked_Off,
		SF_TwoHandControlTypeII_State#Locked_On:
			Ready := TRUE;
			S_TwoHandOut := SAFEBOOL_Constant#SAFEFALSE;
			SafetyDemand := TRUE;
			Error := FALSE;
		SF_TwoHandControlTypeII_State#Error_B1,
		SF_TwoHandControlTypeII_State#Error_B2,
		SF_TwoHandControlTypeII_State#Error_B1_and_B2:
			Ready := TRUE;
			S_TwoHandOut := SAFEBOOL_Constant#SAFEFALSE;
			SafetyDemand := FALSE;
			Error := TRUE;
		ELSE
			ENO := FALSE;
	END_CASE;

	ENO := ENO AND CheckSAFEBOOL(S_Button1) AND CheckSAFEBOOL(S_Button2);

END_FUNCTION_BLOCK

END_NAMESPACE
END_NAMESPACE

(* ---- SF_TwoHandControlTypeIII.iecst ---- *)
USING logicals.web.standard.safe;

NAMESPACE logicals.web.standard.safe
NAMESPACE plcopen

TYPE
	SF_TwoHandControlTypeIII_State : UINT(
	/* S_Button1 was TRUE on FB activation. */
	Error_1_B1 := 16#C010,
	/* S_Button2 was TRUE on FB activation. */
	Error_1_B2 := 16#C020,
	/* The signals at S_Button1 and S_Button2 were TRUE on FB activation. */
	Error_1_B1_and_B2 := 16#C030,
	/* S_Button1 was FALSE and S_Button 2 was TRUE after 500 ms in state 8005. */
	Error_2_B1 := 16#C040,
	/* S_Button1 was TRUE and S_Button 2 was FALSE after 500 ms in state 8005. */
	Error_2_B2 := 16#C050,
	/* S_Button1 was TRUE and S_Button 2 was TRUE after 500 ms in state 8005 or 8006.
	 * This state is only possible when the states of the inputs (S_Button1 and S_Button2)
	 * change from divergent to convergent (both TRUE) simultaneously when the timer elapses (500 ms) at the same cycle.
	 */
	Error_2_B1_and_B2 := 16#C060,
	/* The function block is not active (initial state). */
	Idle := 16#0000,
	/* Both buttons actuated correctly. The safety related output is enabled. */
	Buttons_Actuated := 16#8000,
	/* Function block is active, but in the Init state. */
	Init := 16#8001,
	/* No Button is actuated. */
	Buttons_Released := 16#8802,
	/* Only Button 1 is actuated. Start monitoring timer. */
	Button_1_Actuated := 16#8804,
	/* Only Button 2 is actuated. Start monitoring timer. */
	Button_2_Actuated := 16#8806,
	/* The safety related output was enabled and is disabled again.
	 * FALSE at both S_Button1 and S_Button2 was not achieved after disabling the safety related output.
	 * In this state, S_Button1 is TRUE and S_Button2 is FALSE after disabling the safety related output.
	 */
	Button_2_Released := 16#8808,
	/* The safety related output was enabled and is disabled again.
	 * FALSE at both S_Button1 and S_Button2 was not achieved after disabling the safety related output.
	 * In this state, S_Button1 is FALSE and S_Button2 is TRUE after disabling the safety related output.
	 */
	Button_1_Released := 16#880A,
	/* The safety related output was enabled and is disabled again.
	 * FALSE at both S_Button1 and S_Button2 was not achieved after disabling the safety related output.
	 * In this state, S_Button1 is TRUE and S_Button2 is TRUE after disabling the safety related output.
	 */
	Locked_Off := 16#880C,
	/* Incorrect actuation of the buttons. Waiting for release of both buttons. */
	Locked_On := 16#880E
	);
END_TYPE

/*
 * This function block provides the two-hand control functionality for type III A, B and C.
 * The difference is in the input processing of the switches (single contact, 2 switches per input (equivalent),
 * 2 switches per input (antivalent). (see EN 574, Section 4 Type III. Fixed specified time difference is 500 ms).
 */
FUNCTION_BLOCK SF_TwoHandControlTypeIII
	{ altName:="SF_TwoHandControlTypeIII"; bgColor:="Gold"; width:=420; }
	VAR_INPUT
		/* See Section 5.1.1 General Input Parameters */
		Activate : BOOL := FALSE;
		/* Variable.
		 * Input of button 1 (for category 3 or 4: two antivalent contacts)
		 * FALSE: Button 1 released.
		 * TRUE: Button 1 actuated. */
		S_Button1 : SAFEBOOL := SAFEBOOL_Constant#SAFEFALSE;
		/* Variable.
		 * Input of button 2 (for category 3 or 4: two antivalent contacts)
		 * FALSE: Button 2 released.
		 * TRUE: Button 2 actuated. */
		S_Button2 : SAFEBOOL := SAFEBOOL_Constant#SAFEFALSE;
	END_VAR
	VAR_OUTPUT
		/* See Section 5.1.2 General Output Parameters */
		Ready : BOOL := FALSE;
		/* Safety related output signal.
		 * FALSE: No correct two hand operation.
		 * TRUE: S_Button1 and S_Button2 inputs changed from FALSE to TRUE within 500 ms and no error occurred.
		 * The two hand operation has been performed correctly. */
		S_TwoHandOut : SAFEBOOL := FALSE;
		/* Optional. See 5.1.2 General Output Parameters */
		SafetyDemand : BOOL := FALSE;
		/* See Section 5.1.2 General Output Parameters */
		Error : BOOL := FALSE;
		/* See Section 5.1.2 General Output Parameters */
		DiagCode : WORD := 16#0000;
	END_VAR
	VAR
		Timer : TON;
	END_VAR

	IF(NOT Activate) THEN
		DiagCode := TO_WORD(SF_TwoHandControlTypeIII_State#Idle);
	ELSE
		CASE TO_UINT(DiagCode) OF
			SF_TwoHandControlTypeIII_State#Idle:
				/* IF(Activate) THEN - Active is always true here */
					DiagCode := TO_WORD(SF_TwoHandControlTypeIII_State#Init);
			SF_TwoHandControlTypeIII_State#Init:
				IF(IS(S_Button1)) AND (IS_NOT(S_Button2)) THEN
					DiagCode := TO_WORD(SF_TwoHandControlTypeIII_State#Error_1_B1);
				ELSIF (IS_NOT(S_Button1)) AND (IS(S_Button2)) THEN
					DiagCode := TO_WORD(SF_TwoHandControlTypeIII_State#Error_1_B2);
				ELSIF (IS(S_Button1)) AND (IS(S_Button2)) THEN
					DiagCode := TO_WORD(SF_TwoHandControlTypeIII_State#Error_1_B1_and_B2);
				ELSE /* (IS_NOT(S_Button1)) AND (IS_NOT(S_Button2)) THEN */
					DiagCode := TO_WORD(SF_TwoHandControlTypeIII_State#Buttons_Released);
				END_IF;
			SF_TwoHandControlTypeIII_State#Error_1_B1:
				IF(IS_NOT(S_Button1)) AND (IS_NOT(S_Button2)) THEN
					DiagCode := TO_WORD(SF_TwoHandControlTypeIII_State#Buttons_Released);
				END_IF;
			SF_TwoHandControlTypeIII_State#Error_1_B2:
				IF(IS_NOT(S_Button1)) AND (IS_NOT(S_Button2)) THEN
					DiagCode := TO_WORD(SF_TwoHandControlTypeIII_State#Buttons_Released);
				END_IF;
			SF_TwoHandControlTypeIII_State#Error_1_B1_and_B2:
				IF(IS_NOT(S_Button1)) AND (IS_NOT(S_Button2)) THEN
					DiagCode := TO_WORD(SF_TwoHandControlTypeIII_State#Buttons_Released);
				END_IF;
			SF_TwoHandControlTypeIII_State#Buttons_Released:
				IF(IS(S_Button1)) AND (IS(S_Button2)) THEN
					DiagCode := TO_WORD(SF_TwoHandControlTypeIII_State#Buttons_Actuated);
				ELSIF(IS(S_Button1)) THEN
					DiagCode := TO_WORD(SF_TwoHandControlTypeIII_State#Button_1_Actuated);
				ELSIF(IS(S_Button2)) THEN
					DiagCode := TO_WORD(SF_TwoHandControlTypeIII_State#Button_2_Actuated);
				END_IF;
			SF_TwoHandControlTypeIII_State#Locked_On:
				IF(IS_NOT(S_Button1)) AND (IS_NOT(S_Button2)) THEN
					DiagCode := TO_WORD(SF_TwoHandControlTypeIII_State#Buttons_Released);
				END_IF;
			SF_TwoHandControlTypeIII_State#Error_2_B1:
				IF(IS_NOT(S_Button1)) AND (IS_NOT(S_Button2)) THEN
					DiagCode := TO_WORD(SF_TwoHandControlTypeIII_State#Buttons_Released);
				END_IF;
			SF_TwoHandControlTypeIII_State#Error_2_B2:
				IF(IS_NOT(S_Button1)) AND (IS_NOT(S_Button2)) THEN
					DiagCode := TO_WORD(SF_TwoHandControlTypeIII_State#Buttons_Released);
				END_IF;
			SF_TwoHandControlTypeIII_State#Error_2_B1_and_B2:
				IF(IS_NOT(S_Button1)) AND (IS_NOT(S_Button2)) THEN
					DiagCode := TO_WORD(SF_TwoHandControlTypeIII_State#Buttons_Released);
				END_IF;
			SF_TwoHandControlTypeIII_State#Button_2_Actuated:
				Timer();
				IF(Timer.Q) THEN
					IF(IS(S_Button1)) AND (IS(S_Button2)) THEN
						DiagCode := TO_WORD(SF_TwoHandControlTypeIII_State#Error_2_B1_and_B2);
					ELSE
						DiagCode := TO_WORD(SF_TwoHandControlTypeIII_State#Error_2_B1);
					END_IF;
				ELSIF(IS_NOT(S_Button1)) AND (IS_NOT(S_Button2)) THEN
					DiagCode := TO_WORD(SF_TwoHandControlTypeIII_State#Buttons_Released);
				ELSIF(IS(S_Button1)) AND (IS_NOT(S_Button2)) THEN
					DiagCode := TO_WORD(SF_TwoHandControlTypeIII_State#Locked_On);
				ELSIF(IS(S_Button1)) AND (IS(S_Button2)) THEN
					DiagCode := TO_WORD(SF_TwoHandControlTypeIII_State#Buttons_Actuated);
				END_IF;
			SF_TwoHandControlTypeIII_State#Button_1_Actuated:
				Timer();
				IF(Timer.Q) THEN
					IF(IS(S_Button1)) AND (IS(S_Button2)) THEN
						DiagCode := TO_WORD(SF_TwoHandControlTypeIII_State#Error_2_B1_and_B2);
					ELSE
						DiagCode := TO_WORD(SF_TwoHandControlTypeIII_State#Error_2_B2);
					END_IF;
				ELSIF(IS_NOT(S_Button1)) AND (IS_NOT(S_Button2)) THEN
					DiagCode := TO_WORD(SF_TwoHandControlTypeIII_State#Buttons_Released);
				ELSIF(IS_NOT(S_Button1)) AND (IS(S_Button2)) THEN
					DiagCode := TO_WORD(SF_TwoHandControlTypeIII_State#Locked_On);
				ELSIF(IS(S_Button1)) AND (IS(S_Button2)) THEN
					DiagCode := TO_WORD(SF_TwoHandControlTypeIII_State#Buttons_Actuated);
				END_IF;
			SF_TwoHandControlTypeIII_State#Locked_Off:
				IF(IS_NOT(S_Button1)) AND (IS(S_Button2)) THEN
					DiagCode := TO_WORD(SF_TwoHandControlTypeIII_State#Button_1_Released);
				ELSIF(IS(S_Button1)) AND (IS_NOT(S_Button2)) THEN
					DiagCode := TO_WORD(SF_TwoHandControlTypeIII_State#Button_2_Released);
				ELSIF(IS_NOT(S_Button1)) AND (IS_NOT(S_Button2)) THEN
					DiagCode := TO_WORD(SF_TwoHandControlTypeIII_State#Buttons_Released);
				END_IF;
			SF_TwoHandControlTypeIII_State#Button_1_Released:
				IF(IS(S_Button1)) AND (IS(S_Button2)) THEN
					DiagCode := TO_WORD(SF_TwoHandControlTypeIII_State#Locked_Off);
				ELSIF(IS(S_Button1)) AND (IS_NOT(S_Button2)) THEN
					DiagCode := TO_WORD(SF_TwoHandControlTypeIII_State#Button_2_Released);
				ELSIF(IS_NOT(S_Button1)) AND (IS_NOT(S_Button2)) THEN
					DiagCode := TO_WORD(SF_TwoHandControlTypeIII_State#Buttons_Released);
				END_IF;
			SF_TwoHandControlTypeIII_State#Button_2_Released:
				IF(IS(S_Button1)) AND (IS(S_Button2)) THEN
					DiagCode := TO_WORD(SF_TwoHandControlTypeIII_State#Locked_Off);
				ELSIF(IS_NOT(S_Button1)) AND (IS(S_Button2)) THEN
					DiagCode := TO_WORD(SF_TwoHandControlTypeIII_State#Button_1_Released);
				ELSIF(IS_NOT(S_Button1)) AND (IS_NOT(S_Button2)) THEN
					DiagCode := TO_WORD(SF_TwoHandControlTypeIII_State#Buttons_Released);
				END_IF;
			SF_TwoHandControlTypeIII_State#Buttons_Actuated:
				IF(IS(S_Button1)) AND (IS_NOT(S_Button2)) THEN
					DiagCode := TO_WORD(SF_TwoHandControlTypeIII_State#Button_2_Released);
				ELSIF(IS_NOT(S_Button1)) AND (IS(S_Button2)) THEN
					DiagCode := TO_WORD(SF_TwoHandControlTypeIII_State#Button_1_Released);
				ELSIF(IS_NOT(S_Button1)) AND (IS_NOT(S_Button2)) THEN
					DiagCode := TO_WORD(SF_TwoHandControlTypeIII_State#Buttons_Released);
				END_IF;
			ELSE
				ENO := FALSE;
		END_CASE;
	END_IF;

	CASE TO_UINT(DiagCode) OF
		SF_TwoHandControlTypeIII_State#Idle:
			Timer(IN := FALSE);
			Ready := FALSE;
			S_TwoHandOut := SAFEBOOL_Constant#SAFEFALSE;
			SafetyDemand := FALSE;
			Error := FALSE;
		SF_TwoHandControlTypeIII_State#Buttons_Actuated:
			Timer(IN := FALSE);
			Ready := TRUE;
			S_TwoHandOut := SAFEBOOL_Constant#SAFETRUE;
			SafetyDemand := FALSE;
			Error := FALSE;
		SF_TwoHandControlTypeIII_State#Init:
			Timer(IN := FALSE);
			Ready := TRUE;
			S_TwoHandOut := SAFEBOOL_Constant#SAFEFALSE;
			SafetyDemand := FALSE;
			Error := FALSE;
		SF_TwoHandControlTypeIII_State#Buttons_Released,
		SF_TwoHandControlTypeIII_State#Button_2_Released,
		SF_TwoHandControlTypeIII_State#Button_1_Released,
		SF_TwoHandControlTypeIII_State#Locked_Off,
		SF_TwoHandControlTypeIII_State#Locked_On:
			Timer(IN := FALSE);
			Ready := TRUE;
			S_TwoHandOut := SAFEBOOL_Constant#SAFEFALSE;
			SafetyDemand := TRUE;
			Error := FALSE;
		SF_TwoHandControlTypeIII_State#Button_1_Actuated,
		SF_TwoHandControlTypeIII_State#Button_2_Actuated:
			Timer(IN := TRUE, PT := T#500ms);
			Ready := TRUE;
			S_TwoHandOut := SAFEBOOL_Constant#SAFEFALSE;
			SafetyDemand := TRUE;
			Error := FALSE;
		SF_TwoHandControlTypeIII_State#Error_1_B1,
		SF_TwoHandControlTypeIII_State#Error_1_B2,
		SF_TwoHandControlTypeIII_State#Error_1_B1_and_B2,
		SF_TwoHandControlTypeIII_State#Error_2_B1,
		SF_TwoHandControlTypeIII_State#Error_2_B2,
		SF_TwoHandControlTypeIII_State#Error_2_B1_and_B2:
			Timer(IN := FALSE);
			Ready := TRUE;
			S_TwoHandOut := SAFEBOOL_Constant#SAFEFALSE;
			SafetyDemand := FALSE;
			Error := TRUE;
		ELSE
			ENO := FALSE;
	END_CASE;

	ENO := ENO AND CheckSAFEBOOL(S_Button1) AND CheckSAFEBOOL(S_Button2);

END_FUNCTION_BLOCK

END_NAMESPACE
END_NAMESPACE

(* ---- SFB_GenericSafetyDemand.iecst ---- *)
USING logicals.web.standard.safe;

NAMESPACE logicals.web.standard.safe
NAMESPACE plcopen

TYPE
	SFB_GenericSafetyDemand_State : UINT(
	/* Reset is TRUE while waiting for S_SafetyDemandIn = TRUE. */
	Reset_Error_1 := 16#C001,
	/* Reset is TRUE while waiting for S_SafetyDemandIn = TRUE. */
	Reset_Error_2 := 16#C011,
	/* The function block is not active (initial state). */
	Idle := 16#0000,
	/* Activation is TRUE. The function block was enabled. Check if S_StartReset is required. */
	Init := 16#8001,
	/* Activation is TRUE. Check if Reset is FALSE and wait for S_SafetyDemandIn = TRUE. */
	Wait_for_S_SafetyDemandIn_1 := 16#8802,
	/* Activation is TRUE. S_SafetyDemandIn = TRUE. Wait for rising trigger of Reset. */
	Wait_for_Reset_1 := 16#8402,
	/* Activation is TRUE. Safety demand detected. Check if Reset is FALSE and wait for S_SafetyDemandIn = TRUE. */
	Wait_for_S_SafetyDemandIn_2 := 16#8804,
	/* Activation is TRUE. S_SafetyDemandIn = TRUE. Check for S_AutoReset or wait for rising trigger of Reset. */
	Wait_for_Reset_2 := 16#8404,
	/* Activation is TRUE. S_SafetyDemandIn = TRUE. Functional mode with S_SafetyDemandOut = TRUE. */
	Safety_Output_Enabled := 16#8000
	);
END_TYPE

FUNCTION_BLOCK SFB_GenericSafetyDemand /* is a private module! */
	VAR_INPUT
		/* See Section 5.1.1 General Input Parameters */
		Activate : BOOL := FALSE;
		/* Safety demand input.
		 * Variable.
		 * FALSE: Demand for safety-related response
		 * TRUE: No demand for safety-related response
		 */
		S_SafetyDemandIn : SAFEBOOL := SAFEBOOL_Constant#SAFEFALSE;
		/* See Section 5.1.1 General Input Parameters */
		S_StartReset : SAFEBOOL := SAFEBOOL_Constant#SAFEFALSE;
		/* See Section 5.1.1 General Input Parameters */
		S_AutoReset : SAFEBOOL := SAFEBOOL_Constant#SAFEFALSE;
		/* See Section 5.1.1 General Input Parameters */
		Reset : BOOL := FALSE;
	END_VAR
	VAR_OUTPUT
		/* See Section 5.1.2 General Output Parameters */
		Ready : BOOL := FALSE;
		/* Output for the safety-related response.
		 * FALSE: Safety output disabled. Demand for safety-related response
		 * TRUE: Safety output enabled. No demand for safety-related response
		 */
		S_SafetyDemandOut : SAFEBOOL := SAFEBOOL_Constant#SAFEFALSE;
		/* Optional. See 5.1.2 General Output Parameters */
		SafetyDemand : BOOL := FALSE;
		/* Optional. See 5.1.2 General Output Parameters */
		ResetRequest : BOOL := FALSE;
		/* See Section 5.1.2 General Output Parameters */
		Error : BOOL := FALSE;
		/* See Section 5.1.2 General Output Parameters */
		DiagCode : WORD := 16#0000;
	END_VAR

	IF(NOT Activate) THEN
		DiagCode := TO_WORD(SFB_GenericSafetyDemand_State#Idle);
	ELSE
		CASE TO_UINT(DiagCode) OF
			SFB_GenericSafetyDemand_State#Idle:
				/* IF(Activate) THEN - Active is always true here */
					DiagCode := TO_WORD(SFB_GenericSafetyDemand_State#Init);
			SFB_GenericSafetyDemand_State#Init:
				IF(IS_NOT(S_StartReset)) THEN
					DiagCode := TO_WORD(SFB_GenericSafetyDemand_State#Wait_for_S_SafetyDemandIn_1);
				ELSIF(IS(S_StartReset) AND IS_NOT(S_SafetyDemandIn)) THEN
					DiagCode := TO_WORD(SFB_GenericSafetyDemand_State#Wait_for_S_SafetyDemandIn_2);
				ELSE /* (IS(S_SafetyDemandIn) AND IS(S_StartReset)) THEN */
					DiagCode := TO_WORD(SFB_GenericSafetyDemand_State#Safety_Output_Enabled);
				END_IF;
			SFB_GenericSafetyDemand_State#Wait_for_S_SafetyDemandIn_1:
				IF(IS(S_SafetyDemandIn)) THEN
					IF(Reset) THEN
						DiagCode := TO_WORD(SFB_GenericSafetyDemand_State#Reset_Error_1);
					ELSE
						DiagCode := TO_WORD(SFB_GenericSafetyDemand_State#Wait_for_Reset_1);
					END_IF;
				END_IF;
			SFB_GenericSafetyDemand_State#Wait_for_Reset_1:
				IF(IS_NOT(S_SafetyDemandIn)) THEN
					DiagCode := TO_WORD(SFB_GenericSafetyDemand_State#Wait_for_S_SafetyDemandIn_1);
				ELSIF(Reset) THEN
					DiagCode := TO_WORD(SFB_GenericSafetyDemand_State#Safety_Output_Enabled);
				END_IF;
			SFB_GenericSafetyDemand_State#Reset_Error_1:
				IF(NOT Reset) THEN
					DiagCode := TO_WORD(SFB_GenericSafetyDemand_State#Wait_for_Reset_1);
				END_IF;
			SFB_GenericSafetyDemand_State#Wait_for_S_SafetyDemandIn_2:
				IF (IS(S_SafetyDemandIn)) THEN
					IF(Reset) THEN
						DiagCode := TO_WORD(SFB_GenericSafetyDemand_State#Reset_Error_2);
					ELSIF(IS_NOT(S_AutoReset)) THEN
						DiagCode := TO_WORD(SFB_GenericSafetyDemand_State#Wait_for_Reset_2);
					ELSIF(IS(S_AutoReset)) THEN
						DiagCode := TO_WORD(SFB_GenericSafetyDemand_State#Safety_Output_Enabled);
					END_IF;
				END_IF;
			SFB_GenericSafetyDemand_State#Wait_for_Reset_2:
				IF(IS_NOT(S_SafetyDemandIn)) THEN
					DiagCode := TO_WORD(SFB_GenericSafetyDemand_State#Wait_for_S_SafetyDemandIn_2);
				ELSIF(Reset OR IS(S_AutoReset)) THEN
					DiagCode := TO_WORD(SFB_GenericSafetyDemand_State#Safety_Output_Enabled);
				END_IF;
			SFB_GenericSafetyDemand_State#Reset_Error_2:
				IF(NOT Reset) THEN
					DiagCode := TO_WORD(SFB_GenericSafetyDemand_State#Wait_for_Reset_2);
				END_IF;
			SFB_GenericSafetyDemand_State#Safety_Output_Enabled:
				IF(IS_NOT(S_SafetyDemandIn)) THEN
					DiagCode := TO_WORD(SFB_GenericSafetyDemand_State#Wait_for_S_SafetyDemandIn_2);
				END_IF;
			ELSE
				ENO := FALSE;
		END_CASE;
	END_IF;

	CASE TO_UINT(DiagCode) OF
		SFB_GenericSafetyDemand_State#Idle:
			Ready := FALSE;
			S_SafetyDemandOut := SAFEBOOL_Constant#SAFEFALSE;
			SafetyDemand := FALSE;
			ResetRequest := FALSE;
			Error := FALSE;
		SFB_GenericSafetyDemand_State#Init:
			Ready := TRUE;
			S_SafetyDemandOut := SAFEBOOL_Constant#SAFEFALSE;
			SafetyDemand := FALSE;
			ResetRequest := FALSE;
			Error := FALSE;
		SFB_GenericSafetyDemand_State#Wait_for_S_SafetyDemandIn_1, SFB_GenericSafetyDemand_State#Wait_for_S_SafetyDemandIn_2:
			Ready := TRUE;
			S_SafetyDemandOut := SAFEBOOL_Constant#SAFEFALSE;
			SafetyDemand := TRUE;
			ResetRequest := FALSE;
			Error := FALSE;
		SFB_GenericSafetyDemand_State#Wait_for_Reset_1, SFB_GenericSafetyDemand_State#Wait_for_Reset_2:
			Ready := TRUE;
			S_SafetyDemandOut := SAFEBOOL_Constant#SAFEFALSE;
			SafetyDemand := FALSE;
			ResetRequest := TRUE;
			Error := FALSE;
		SFB_GenericSafetyDemand_State#Safety_Output_Enabled:
			Ready := TRUE;
			S_SafetyDemandOut := SAFEBOOL_Constant#SAFETRUE;
			SafetyDemand := FALSE;
			ResetRequest := FALSE;
			Error := FALSE;
		SFB_GenericSafetyDemand_State#Reset_Error_1, SFB_GenericSafetyDemand_State#Reset_Error_2:
			Ready := TRUE;
			S_SafetyDemandOut := SAFEBOOL_Constant#SAFEFALSE;
			SafetyDemand := FALSE;
			ResetRequest := FALSE;
			Error := TRUE;
		ELSE
			ENO := FALSE;
	END_CASE;

	ENO := ENO AND CheckSAFEBOOL(S_SafetyDemandIn) AND CheckSAFEBOOL(S_StartReset) AND CheckSAFEBOOL(S_AutoReset);

END_FUNCTION_BLOCK

END_NAMESPACE
END_NAMESPACE
